SUBAPPLICATION Blink_Knickdeichsel_heben (* Subapplication Type *)
  (* Standard: 61499-2 *)
  (* Version 1.0, 2023-02-11, franz *)
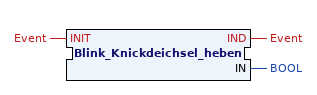
  EVENT_INPUT
    INIT;
  END_EVENT
  EVENT_OUTPUT
    IND;
  END_EVENT
  VAR_OUTPUT
    IN : BOOL;
  END_VAR
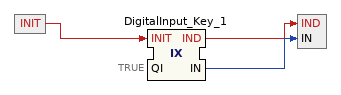
  FBS
    DigitalInput_Key_1 : IX(QI := TRUE);
  END_FBS
  EVENT_CONNECTIONS
    INIT TO DigitalInput_Key_1.INIT;
    DigitalInput_Key_1.IND TO IND;
  END_CONNECTIONS
  DATA_CONNECTIONS
    DigitalInput_Key_1.IN TO IN;
  END_CONNECTIONS
END_SUBAPPLICATION
